{attribute 'GeneratedUsingTerminal: EL3161-0000-0016'}
{attribute addProperty BoxType "EL3161-0000-0016"}
{attribute addProperty Id "AI_StandardAT %I*AI_Standard_A8DF64E310WcStateAT %I*WcState_9091E0EB2InfoDataAT %I*InfoData_32EB74EA10"}
{attribute addProperty CRC "2916756744"}
{attribute addProperty Size "22"}
TYPE EL3161_ADDA2D08 EXTENDS EtcSlaveTerminalBase_947E5A46 :
STRUCT
	{attribute addProperty Name "AI_Standard"}
	AI_Standard : AI_Standard_A8DF64E3;
	{attribute addProperty Name "WcState"}
	WcState : WcState_9091E0EB;
	{attribute addProperty Name "InfoData"}
	InfoData : InfoData_32EB74EA;
END_STRUCT
END_TYPE

(* stored: Version 1.2.0.0, ProductVersion 3.1.4024.9
   DUT EL3161_ADDA2D08: Id {dcc606da-3a5b-475a-9918-00699eeb0b5c} *)
